TYPE
    Locations :
    STRUCT
        LocX : INT;
        LocY : INT;
        Roll : INT;
    END_STRUCT
END_TYPE

(* stored: Version 1.1.0.1, ProductVersion 3.1.4024.12
   DUT Locations: Id {46d24a07-67ac-08b1-1e38-8227c081cbd4} *)
